Fanuc KAREL source: kc00047.KL

-- PROVISIONAL review KL for V1013-1; original PC SHA256 bdef47e1033e0530f6c10937849021ab3de6c7f7b52b0565584bc57a4f8019fb
-- Incomplete behavior may be omitted. Consult companion uncertainty JSON. Do not deploy.
PROGRAM KC00047
%NOLOCKGROUP
BEGIN
  -- UNRESOLVED_PC offsets 5-27; opcodes 27,22,22,22,31
  -- UNRESOLVED_PC offsets 32-36; opcodes 7F
END KC00047
